PROGRAM MAIN
VAR
END_VAR

Plc_Prog();

END_PROGRAM

(* stored: Version 1.1.0.1, ProductVersion 3.1.4024.9
   POU MAIN: Id {814f1b37-eda7-4e96-b2f6-66e7ed32dd0e}, SpecialFunc None *)
